(* Logix 5000 project; controller parts_sorting_system vendor 1 type 14 code 196 rev 36.11; software revision 36.00 *)

TASK MainTask (continuous, watchdog 500 ms) : MainProgram

MODULES
   Local : vendor 1 type 14 code 196 (5069 0, rev 36.11)
END_MODULES

VAR_GLOBAL   (* controller tags *)
   Conveyor_Run : BOOL;   // Simulated conveyor motor run
   PB_Reset : BOOL;   // system reset pushbutton
   PB_Start : BOOL := 1;   // start push button
   PB_stop : BOOL;   // stop pushbutton
   PE_Entry : BOOL;   // entry photoeye detects a new part
   Reject_Gate : BOOL;   // reject/diverter actuator output
   Vision_Bad : BOOL;   // simulated vision result, 1 = bad, 0 = good
END_VAR

PROGRAM MainProgram   (* main routine MainRoutine *)
VAR
   Bad_At_Reject : BOOL;   // Indicates tracked bad bit at reject station
   BadPartTrack : DINT[1];   // tracks bad part
   BSL_Bad_Control : CONTROL := (LEN := 10);   // Control structure for bad-part shift register
   BSL_Present_Control : CONTROL := (LEN := 10);   // Control structure for part-present shift register
   C_BadParts : COUNTER := (PRE := 9999);
   C_GoodParts : COUNTER := (PRE := 9999);   // counts all good parts
   C_RejectedParts : COUNTER;   // counts rejected bad parts
   C_RejectParts : COUNTER;   // counts all bad parts
   C_TotalParts : COUNTER := (PRE := 9999);   // counts all parts entering
   Conveyor_Run : BOOL;   // Simulated conveyor motor run
   Entry_Event : BOOL;   // One-shot pulse for new part entry
   Load_Badbit : BOOL;   // Bit loaded into bad-part register
   Load_PresentBit : BOOL;   // Bit loaded into part-present register
   Manual_Step_Pulse : BOOL;   // One-scan manual pulse
   ONS_Enrty : BOOL;   // storage bit for entry sensor one-shot
   ONS_RejectCount : BOOL;   // Storage bit for rejected counter one-shot
   ONS_Shift : BOOL;   // Storage bit for conveyor pulse one-shot
   ONS_Step : BOOL;   // One-shot storage
   Part_At_Reject : BOOL;   // indicates tracked part at reject station
   PartPresentTrack : DINT[1];   // Tracks physical part location
   PB_Reset : BOOL;   // system reset pushbutton
   PB_Start : BOOL;   // start push button
   PB_step : BOOL;   // Manual shift pushbutton
   PB_stop : BOOL;   // stop pushbutton
   PE_Entry : BOOL;   // entry photoeye detects a new part
   Reject_Gate : BOOL;   // reject/diverter actuator output
   Reject_Request : BOOL;   // Internal request to fire reject gate
   Shift_Pulse : BOOL;   // One-shot conveyor movement pulse
   System_Run : BOOL;   // master run bit
   T_Pulse : TIMER := (PRE := 500);   // Conveyor pulse generator
   T_Reject : TIMER := (PRE := 300);   // Reject gate pulse timer
   Vision_Bad : BOOL;   // simulated vision result, 1 = bad, 0 = good
END_VAR

ROUTINE MainRoutine   (* ladder *)
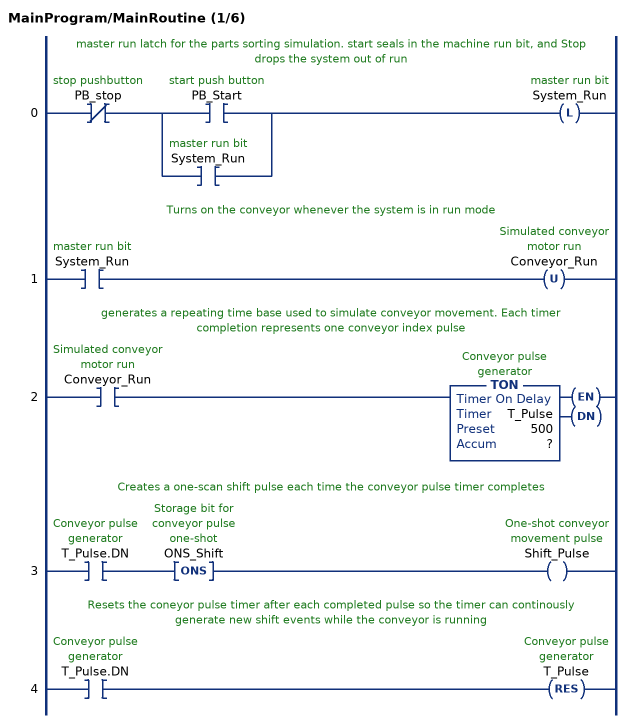
   // master run latch for the parts sorting simulation. start seals in the machine run bit, and Stop drops the system out of run
   0: XIO(PB_stop)[XIC(PB_Start) ,XIC(System_Run) ]OTL(System_Run);
   // Turns on the conveyor whenever the system is in run mode
   1: XIC(System_Run)OTU(Conveyor_Run);
   // generates a repeating time base used to simulate conveyor movement. Each timer completion represents one conveyor index pulse
   2: XIC(Conveyor_Run)TON(T_Pulse,?,?);
   // Creates a one-scan shift pulse each time the conveyor pulse timer completes
   3: XIC(T_Pulse.DN)ONS(ONS_Shift)OTE(Shift_Pulse);
   // Resets the coneyor pulse timer after each completed pulse so the timer can continously generate new shift events while the conveyor is running
   4: XIC(T_Pulse.DN)RES(T_Pulse);
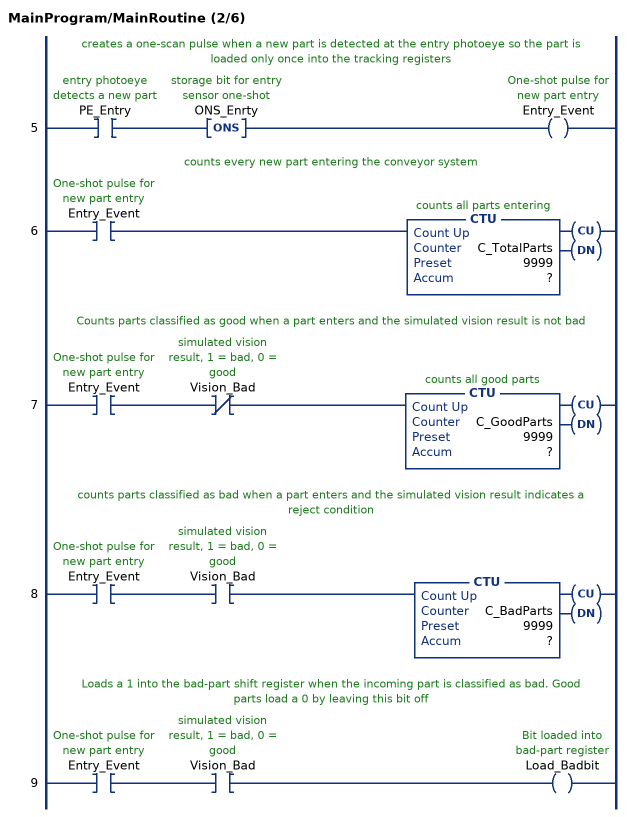
   // creates a one-scan pulse when a new part is detected at the entry photoeye so the part is loaded only once into the tracking registers
   5: XIC(PE_Entry)ONS(ONS_Enrty)OTE(Entry_Event);
   // counts every new part entering the conveyor system
   6: XIC(Entry_Event)CTU(C_TotalParts,?,?);
   // Counts parts classified as good when a part enters and the simulated vision result is not bad
   7: XIC(Entry_Event)XIO(Vision_Bad)CTU(C_GoodParts,?,?);
   // counts parts classified as bad when a part enters and the simulated vision result indicates a reject condition
   8: XIC(Entry_Event)XIC(Vision_Bad)CTU(C_BadParts,?,?);
   // Loads a 1 into the bad-part shift register when the incoming part is classified as bad. Good parts load a 0 by leaving this bit off
   9: XIC(Entry_Event)XIC(Vision_Bad)OTE(Load_Badbit);
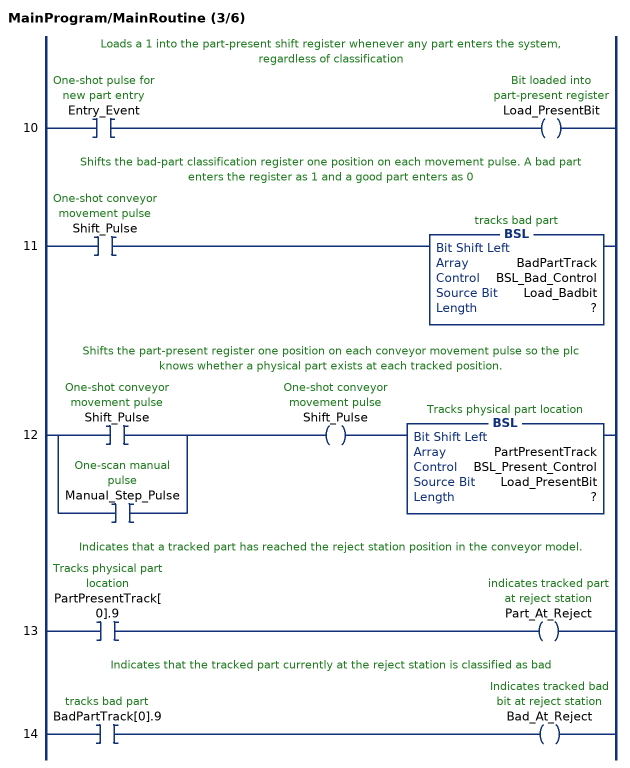
   // Loads a 1 into the part-present shift register whenever any part enters the system, regardless of classification
   10: XIC(Entry_Event)OTE(Load_PresentBit);
   // Shifts the bad-part classification register one position on each movement pulse. A bad part enters the register as 1 and a good part enters as 0
   11: XIC(Shift_Pulse)BSL(BadPartTrack,BSL_Bad_Control,Load_Badbit,?);
   // Shifts the part-present register one position on each conveyor movement pulse so the plc knows whether a physical part exists at each tracked position.
   12: [XIC(Shift_Pulse) ,XIC(Manual_Step_Pulse) ]OTE(Shift_Pulse)BSL(PartPresentTrack,BSL_Present_Control,Load_PresentBit,?);
   // Indicates that a tracked part has reached the reject station position in the conveyor model.
   13: XIC(PartPresentTrack[0].9)OTE(Part_At_Reject);
   // Indicates that the tracked part currently at the reject station is classified as bad
   14: XIC(BadPartTrack[0].9)OTE(Bad_At_Reject);
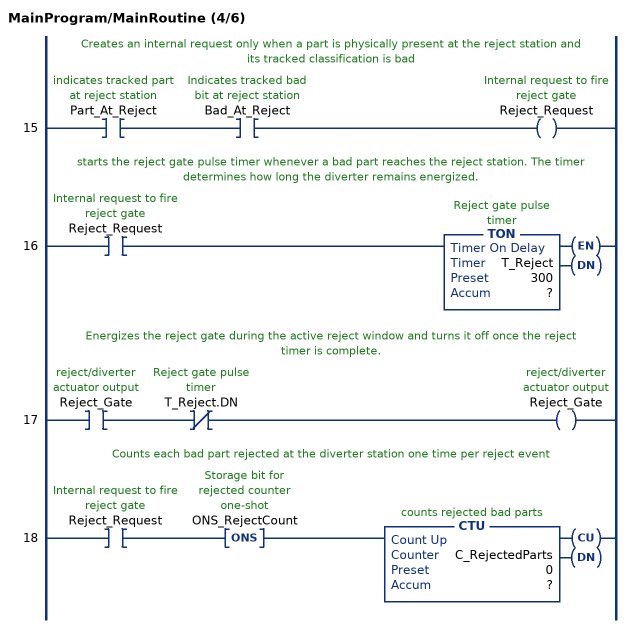
   // Creates an internal request only when a part is physically present at the reject station and its tracked classification is bad
   15: XIC(Part_At_Reject)XIC(Bad_At_Reject)OTE(Reject_Request);
   // starts the reject gate pulse timer whenever a bad part reaches the reject station. The timer determines how long the diverter remains energized.
   16: XIC(Reject_Request)TON(T_Reject,?,?);
   // Energizes the reject gate during the active reject window and turns it off once the reject timer is complete.
   17: XIC(Reject_Gate)XIO(T_Reject.DN)OTE(Reject_Gate);
   // Counts each bad part rejected at the diverter station one time per reject event
   18: XIC(Reject_Request)ONS(ONS_RejectCount)CTU(C_RejectedParts,?,?);
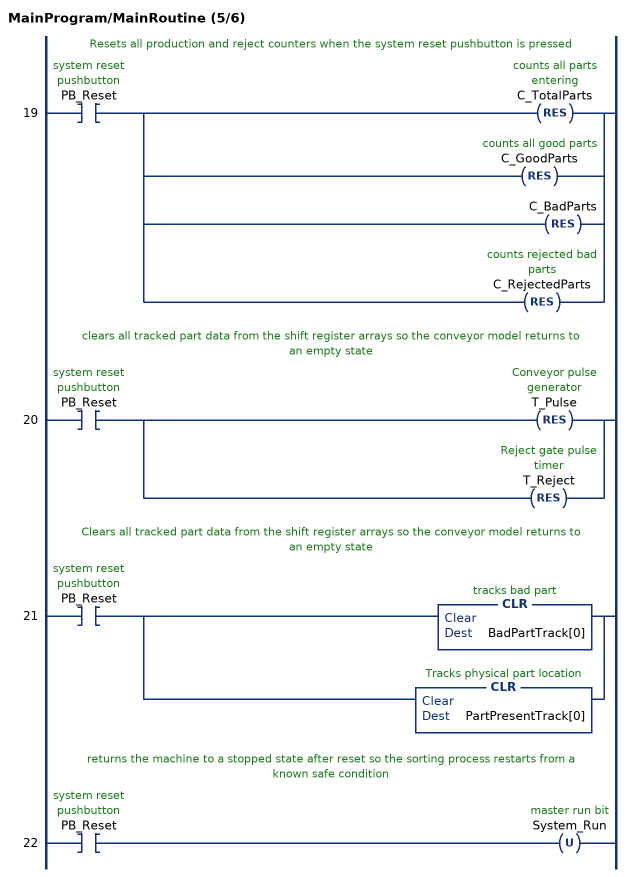
   // Resets all production and reject counters when the system reset pushbutton is pressed
   19: XIC(PB_Reset)[RES(C_TotalParts) ,RES(C_GoodParts) ,RES(C_BadParts) ,RES(C_RejectedParts) ];
   // clears all tracked part data from the shift register arrays so the conveyor model returns to an empty state
   20: XIC(PB_Reset)[RES(T_Pulse) ,RES(T_Reject) ];
   // Clears all tracked part data from the shift register arrays so the conveyor model returns to an empty state
   21: XIC(PB_Reset)[CLR(BadPartTrack[0]) ,CLR(PartPresentTrack[0]) ];
   // returns the machine to a stopped state after reset so the sorting process restarts from a known safe condition
   22: XIC(PB_Reset)OTU(System_Run);
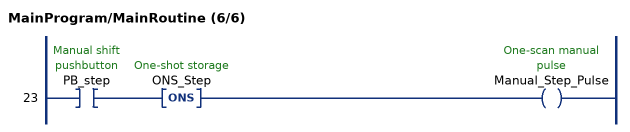
   23: XIC(PB_step)ONS(ONS_Step)OTE(Manual_Step_Pulse);
END_ROUTINE
END_PROGRAM
